(* IEC 61131-3 sources: ml2plc/examples/models/structured_text (part 2) *)

(* ---- test10_5k.st ---- *)
FUNCTION_BLOCK NeuralNetworkFB

VAR_INPUT
    input_data : ARRAY[0..4] OF REAL;
END_VAR

VAR_OUTPUT
    output_data : ARRAY[0..2] OF REAL;
END_VAR

VAR CONSTANT
    weights_0 : ARRAY[0..109] OF REAL := [-0.235502, 0.374035, 0.029982, 0.212839, 0.258987, -0.111841, 0.244708, -0.308510, 0.228488, 0.160992, 0.383056, 0.408669, -0.403928, -0.237195, 0.098766, -0.443759, -0.297004, -0.183076, 0.183679, -0.150052, -0.244251, -0.296679, 0.282903, -0.114856, -0.204128, 0.239042, -0.264883, 0.227759, -0.321238, 0.035633, 0.262893, -0.322360, -0.104940, 0.452904, 0.456325, 0.030485, -0.030166, -0.158633, 0.107382, -0.069652, -0.001856, -0.272029, -0.007177, -0.122300, 0.214300, 0.062439, 0.300184, -0.465629, -0.025417, -0.246331, 0.205803, 0.023458, -0.192963, -0.407002, -0.281354, -0.300315, -0.372232, -0.163916, -0.173461, 0.322071, 0.477836, 0.353802, 0.206684, 0.197231, 0.380607, 0.522870, -0.316586, 0.070922, 0.220201, 0.307742, -0.224637, -0.294651, -0.101183, 0.079923, 0.277857, 0.419958, -0.196677, -0.210945, -0.373816, 0.376826, -0.382129, -0.066666, 0.071888, 0.258300, -0.222091, 0.385427, -0.307561, -0.131309, 0.078177, -0.005495, 0.222825, -0.380124, -0.054474, -0.272398, -0.041792, 0.481035, 0.159107, 0.424615, 0.015366, 0.498193, -0.156387, 0.359789, 0.473488, -0.037305, -0.414866, 0.249786, -0.175640, 0.421966, 0.072167, -0.130746];
    bias_0 : ARRAY[0..21] OF REAL := [0.056635, -0.124397, -0.266900, -0.117066, -0.247369, -0.074615, -0.135742, 0.004444, -0.217433, -0.099763, 0.119883, -0.049615, -0.077851, -0.192466, -0.024998, 0.047683, 0.188981, -0.322050, 0.077329, -0.218410, -0.089648, -0.137956];

    weights_1 : ARRAY[0..483] OF REAL := [0.079049, -0.347925, 0.337554, -0.033540, 0.138506, 0.092452, -0.378136, 0.249819, -0.085962, 0.006912, 0.181653, 0.205352, -0.241950, 0.184875, 0.065784, -0.124519, 0.197723, 0.064407, 0.105942, 0.236089, 0.209018, 0.178479, 0.218949, -0.102088, -0.093211, -0.269140, -0.040398, 0.044989, 0.262907, 0.256715, -0.098784, 0.291057, 0.262021, 0.194998, -0.235076, -0.154412, -0.103262, 0.045983, -0.148590, -0.016494, -0.348144, 0.355634, -0.331634, -0.158894, 0.055906, 0.248997, 0.337778, -0.223945, -0.040168, 0.011934, -0.216079, -0.302210, -0.101061, 0.099673, 0.114095, 0.322268, -0.059129, -0.282656, -0.375054, 0.167089, -0.216769, 0.033994, -0.177784, 0.290487, -0.068697, 0.124034, 0.228402, -0.131462, -0.027060, 0.223431, -0.392828, 0.256138, -0.026546, 0.114889, -0.114368, 0.116107, -0.211801, 0.206436, 0.112972, 0.212281, -0.293026, -0.028103, 0.086852, -0.201455, -0.398612, 0.019805, 0.232748, 0.214277, -0.045702, -0.094083, -0.236141, 0.221850, 0.089407, -0.034819, -0.354278, 0.161435, 0.190216, 0.158098, 0.228709, -0.163889, 0.277531, -0.243516, 0.211692, -0.334966, 0.207670, 0.204391, 0.121696, -0.322424, 0.116413, -0.058254, -0.120124, -0.065694, 0.240498, -0.015988, -0.299633, 0.134494, -0.267642, -0.028926, 0.145824, -0.105526, -0.245366, -0.248820, 0.101097, -0.096212, -0.271919, -0.017597, -0.037329, 0.021210, -0.182566, 0.064379, -0.230258, -0.351002, -0.238026, 0.179422, 0.348074, -0.171654, 0.183988, -0.129054, -0.097976, 0.232130, 0.159159, -0.230301, 0.177287, -0.012360, -0.310712, -0.222650, 0.224205, -0.184178, 0.288744, 0.156265, -0.125907, 0.356347, -0.052188, -0.151564, -0.050163, -0.188746, 0.207031, 0.244088, 0.237136, -0.288542, 0.231177, 0.109337, -0.254618, 0.376183, -0.294310, 0.144768, -0.143697, -0.101113, -0.206989, 0.203110, 0.169697, -0.095264, 0.436408, 0.036662, 0.058565, -0.072889, 0.137062, 0.257720, -0.292869, 0.024309, -0.346628, 0.294436, 0.111847, 0.105722, 0.110252, 0.043315, 0.163461, -0.022499, 0.159847, 0.237663, 0.054308, 0.147833, -0.067078, -0.073643, -0.195978, -0.328734, -0.264882, -0.140460, -0.320087, 0.028090, -0.188938, -0.239834, -0.036262, 0.028815, 0.019727, -0.339510, -0.203977, -0.065838, 0.302599, 0.176075, 0.212229, -0.302148, 0.225811, 0.297823, -0.244519, 0.177079, 0.026356, 0.216062, 0.186228, -0.249791, -0.234059, -0.264074, 0.014307, -0.334354, -0.306848, -0.327795, -0.038307, -0.373215, -0.371131, -0.433094, -0.388753, -0.166083, -0.283418, -0.421748, -0.019741, -0.387288, 0.161504, 0.004465, 0.174149, -0.238579, -0.185134, 0.218629, -0.320004, 0.290548, 0.235413, -0.214184, -0.233729, -0.148321, -0.238665, -0.422416, -0.040923, 0.123327, -0.157409, -0.017170, 0.296382, 0.024681, -0.378978, 0.070786, -0.283947, -0.322869, 0.151345, -0.373138, 0.336530, 0.056313, -0.373142, -0.187809, -0.092519, 0.086954, -0.119277, -0.137913, -0.083906, 0.078384, -0.119447, -0.275883, 0.144350, 0.158292, -0.327999, -0.276656, 0.078429, -0.347799, 0.023557, -0.236602, -0.128356, -0.233653, 0.236965, 0.064413, 0.334948, 0.220999, -0.212444, 0.256759, -0.155419, 0.196652, 0.245904, 0.341258, 0.370730, 0.132005, 0.192064, 0.279513, -0.112169, 0.022927, -0.015424, 0.219870, 0.228535, 0.070248, -0.105873, -0.336300, 0.031945, 0.292533, 0.152411, -0.309550, 0.339161, 0.017188, 0.078137, -0.074693, -0.159284, 0.100658, 0.237390, -0.029114, 0.024597, 0.130221, -0.231880, 0.122851, -0.098909, 0.267768, -0.233404, -0.160178, 0.185329, 0.261339, 0.140867, 0.353704, 0.056444, 0.012285, -0.106170, 0.126114, 0.129954, 0.061448, -0.336865, -0.267193, -0.310728, -0.062605, -0.343586, -0.149127, 0.171627, 0.311902, -0.232079, -0.340220, -0.166417, -0.269893, -0.331138, -0.181041, -0.010986, 0.102309, -0.220985, -0.073660, -0.041843, -0.278722, -0.287776, 0.156741, 0.001601, -0.055916, 0.144559, -0.098055, -0.268363, -0.229689, -0.146128, -0.391409, 0.362549, -0.104388, 0.269200, -0.132739, -0.278950, -0.065837, -0.298305, 0.237254, 0.329178, 0.309923, -0.221904, -0.107192, -0.299514, 0.042806, 0.276688, -0.033415, 0.214313, 0.260739, -0.159463, 0.174015, -0.344592, -0.080061, -0.129057, -0.056141, -0.064048, 0.258323, 0.000715, -0.093780, -0.323654, -0.309229, -0.420076, -0.072576, -0.079502, 0.125576, -0.276341, -0.230562, -0.146622, -0.109113, 0.033652, -0.318611, -0.316500, -0.290675, -0.363042, -0.224463, -0.261462, -0.292973, 0.321195, -0.002662, 0.045876, -0.085935, -0.255877, 0.129174, 0.178717, 0.347154, 0.307062, -0.218534, -0.084984, -0.345322, 0.030590, -0.089027, 0.217998, -0.144714, -0.046250, -0.281607, -0.235275, 0.266412, 0.278757, 0.038723, 0.169535, 0.118446, 0.398865, 0.104389, -0.289460, -0.226774, -0.160745, -0.125390, 0.291478, -0.404079, 0.182954, -0.242632, -0.011222, 0.019191, -0.276508, 0.232760, 0.171934, -0.169843, -0.043784, -0.157749, -0.116427, 0.271703, -0.243017, 0.220278, 0.041874, 0.312852, -0.344001, 0.205275, 0.239192, -0.247240, 0.234474, -0.094469, -0.202707, 0.335269, 0.229963, 0.199586, -0.262707, 0.257955, -0.312206, -0.360458, -0.320586, 0.211516, 0.337735, 0.278487, 0.267389, 0.241000, -0.250274, 0.072497, 0.185405, 0.199016];
    bias_1 : ARRAY[0..21] OF REAL := [-0.155419, -0.267332, -0.021124, -0.086635, -0.086491, 0.106494, -0.081331, -0.149528, 0.128646, 0.006162, -0.052589, -0.175140, 0.004669, -0.158592, -0.001915, -0.165681, -0.032700, -0.202270, -0.109741, 0.031299, -0.051547, 0.080420];

    weights_2 : ARRAY[0..483] OF REAL := [-0.082935, 0.327544, 0.254661, -0.021772, 0.201947, 0.305412, 0.081183, 0.318496, 0.143632, -0.205671, 0.060881, -0.296683, 0.233208, -0.132674, -0.267633, 0.297422, -0.148609, 0.024956, -0.328323, 0.249083, 0.322392, 0.251571, -0.079101, 0.041405, -0.094899, -0.052703, -0.228929, -0.173477, 0.309499, -0.298324, -0.328228, 0.191809, 0.211639, 0.175227, -0.291024, -0.241829, -0.227845, 0.359827, -0.173025, -0.185764, -0.281586, -0.131694, -0.345628, -0.036727, -0.163816, -0.334208, -0.132535, 0.173024, 0.224584, -0.343964, -0.252016, -0.342804, 0.081973, 0.110123, 0.056545, -0.049518, 0.216609, -0.092255, -0.220284, 0.153317, -0.178284, 0.077126, -0.381740, 0.041970, 0.118417, -0.290151, 0.228592, -0.343728, 0.081173, 0.186181, 0.042570, -0.032074, -0.347268, 0.039175, 0.205202, -0.321549, -0.104232, -0.302562, -0.251374, 0.314923, 0.045477, -0.033431, -0.386075, 0.012686, 0.125798, -0.210791, -0.393972, -0.352663, 0.300682, 0.233090, 0.060526, 0.143590, 0.215293, 0.298667, 0.050667, 0.195947, 0.172492, 0.286427, -0.276380, -0.344604, -0.295523, -0.000179, 0.252037, 0.155288, 0.180119, -0.282181, -0.368783, 0.259566, -0.153441, -0.230622, 0.294233, -0.076799, -0.375942, -0.345544, -0.163923, 0.044519, -0.319325, 0.221346, -0.132698, -0.127449, 0.026434, -0.149147, -0.076145, -0.306095, -0.253755, -0.312573, 0.021093, -0.181651, -0.290607, 0.083633, -0.150752, 0.006249, -0.298933, 0.333710, 0.325536, -0.222120, 0.278292, 0.100666, -0.085205, -0.356550, 0.185289, 0.084207, 0.177925, -0.233948, -0.031037, 0.031882, -0.276591, -0.200347, -0.265831, -0.171206, -0.121855, -0.272616, 0.106950, 0.267811, 0.144345, -0.141822, 0.314253, -0.139761, 0.326825, -0.240426, 0.203541, 0.224520, -0.346032, 0.054895, 0.171094, 0.049029, -0.116277, -0.143705, 0.283372, -0.025292, -0.333692, -0.302754, 0.050393, 0.194249, -0.151961, 0.190338, -0.155851, -0.230143, -0.286497, 0.344899, 0.024594, 0.079224, -0.023155, 0.030636, 0.121751, 0.115104, -0.101916, -0.335504, -0.111129, -0.103364, 0.171968, -0.336117, 0.022877, 0.127892, -0.135068, -0.122467, -0.396051, 0.145917, -0.006995, 0.381155, -0.271586, 0.211470, 0.293431, 0.054489, 0.267433, 0.043922, -0.036805, -0.139896, -0.059831, 0.220703, 0.157794, -0.123315, -0.004200, -0.389434, -0.119506, 0.234269, -0.144908, -0.325883, 0.023704, -0.203639, 0.025667, 0.011748, 0.296067, 0.257535, 0.341761, 0.013412, -0.246624, -0.031834, 0.012090, -0.022462, 0.387307, -0.315927, 0.135532, -0.106146, -0.208187, -0.077365, 0.210223, -0.164290, 0.117905, -0.141453, -0.062069, 0.078166, 0.197727, -0.315830, -0.359223, -0.000416, 0.153591, 0.293815, -0.088260, -0.024230, 0.338556, 0.085211, -0.209096, 0.270740, 0.266294, 0.103243, 0.280570, 0.004210, 0.174240, 0.393157, -0.136366, -0.322978, -0.000434, 0.228373, -0.258511, 0.179665, -0.222202, 0.114817, 0.119143, 0.073947, -0.261211, 0.292751, 0.027004, -0.307591, 0.184837, -0.129084, -0.067745, -0.033641, 0.037630, -0.078543, -0.085143, -0.098848, -0.030430, 0.187926, -0.058864, -0.145514, -0.132123, 0.143235, 0.158167, 0.062374, 0.066104, 0.019079, 0.251746, -0.122901, 0.164780, -0.194877, 0.219013, -0.242652, -0.214676, -0.076353, -0.249113, 0.221838, 0.199792, 0.181832, -0.230836, -0.109779, 0.133959, -0.036438, -0.249530, 0.199512, -0.095072, 0.093821, 0.071035, 0.061617, -0.279793, -0.201789, 0.187455, 0.018947, 0.050322, 0.008108, -0.046991, 0.306518, -0.327390, -0.138280, 0.116354, -0.106726, 0.207402, -0.069084, -0.132325, -0.310824, -0.166095, 0.230069, -0.389367, 0.254957, 0.026655, -0.361433, -0.138050, 0.059506, 0.152043, -0.028680, 0.287269, 0.153620, -0.085093, 0.109935, -0.100580, -0.031819, 0.185861, 0.392915, -0.032841, 0.080074, 0.306054, 0.027516, -0.379458, 0.256309, -0.393753, 0.001235, -0.319371, 0.251579, 0.125351, 0.073606, -0.082433, -0.161256, -0.069119, -0.211557, -0.294755, -0.267203, -0.224041, -0.309678, -0.351013, 0.121915, -0.248513, 0.271583, 0.124953, 0.201983, 0.198783, 0.099953, 0.131763, -0.286613, -0.229959, -0.150241, 0.379902, -0.322958, 0.278217, 0.239573, -0.287928, 0.336981, 0.176765, 0.110885, 0.159063, 0.293586, 0.322831, -0.086323, -0.214025, -0.030494, -0.146554, 0.020220, 0.070352, -0.005592, 0.164585, -0.044105, -0.015679, 0.194617, 0.231574, -0.021186, -0.312370, 0.146685, 0.363802, -0.404818, 0.063827, -0.091208, 0.104540, 0.112544, 0.225414, 0.426742, 0.164169, -0.015709, 0.332852, 0.015972, 0.245230, -0.030557, -0.123999, -0.129163, -0.298851, -0.172933, 0.228824, 0.231744, 0.039497, 0.270405, -0.303923, 0.058437, -0.216858, 0.034896, 0.123225, -0.159160, -0.288073, -0.040648, -0.108659, -0.092023, 0.054152, -0.387218, 0.163232, 0.184591, 0.243524, -0.138134, -0.341152, 0.046506, -0.346441, -0.281175, -0.387726, 0.123238, -0.300494, 0.237686, -0.045294, -0.331050, -0.130853, -0.231359, 0.222539, -0.205569, -0.347141, -0.176774, 0.238876, -0.010123, -0.432586, -0.172873, -0.266623, -0.267432, -0.083994, -0.348342, 0.095161, -0.382534, -0.225168, -0.199141, 0.018341, -0.198148, 0.198510, 0.236356, -0.289449, 0.075354, -0.175895, -0.114134, 0.042550, -0.277356, -0.088906, -0.080386];
    bias_2 : ARRAY[0..21] OF REAL := [-0.132522, -0.027953, -0.156794, -0.173189, -0.073986, -0.111488, -0.182651, -0.158691, -0.185292, -0.282737, -0.305989, -0.185168, -0.048515, -0.036091, -0.075189, -0.198026, -0.136586, -0.106037, -0.051125, -0.059318, -0.072963, -0.191347];

    weights_3 : ARRAY[0..483] OF REAL := [-0.070963, 0.130692, -0.269850, 0.140810, -0.058719, 0.300814, 0.273362, -0.241552, 0.052187, 0.139223, -0.312618, 0.302189, 0.204637, 0.280806, 0.249241, 0.239799, -0.030181, 0.299634, -0.158570, -0.240536, 0.039247, -0.093849, -0.069672, -0.110026, 0.104300, 0.006270, -0.065404, -0.061827, 0.137584, 0.113450, 0.233291, 0.031230, -0.224060, -0.007959, -0.009959, -0.207101, 0.114770, 0.173167, 0.251814, -0.079727, -0.083826, -0.260188, -0.310279, 0.104744, 0.107125, 0.207032, -0.318996, 0.159255, 0.034373, 0.237722, 0.033715, -0.121734, -0.224087, 0.206738, 0.059584, 0.299180, 0.068442, -0.156955, 0.145228, -0.100454, -0.225023, -0.273292, 0.280308, 0.093051, -0.354356, 0.032969, -0.196454, -0.130776, -0.143975, 0.084145, 0.129234, -0.034169, 0.310125, -0.085513, 0.109817, -0.218289, 0.008993, 0.240534, 0.285099, -0.293260, -0.239596, -0.215456, 0.128503, -0.107708, 0.160487, 0.124243, 0.151635, 0.304328, -0.107218, 0.270742, 0.065129, 0.166662, -0.046038, -0.054938, 0.022022, -0.104007, 0.128583, -0.099885, -0.048699, -0.033328, 0.088990, -0.288285, -0.222791, -0.051723, 0.290322, -0.252797, -0.030634, -0.152525, -0.258451, -0.281153, -0.326554, 0.119863, 0.153369, -0.265971, -0.090043, -0.078578, -0.240882, 0.180207, -0.119918, -0.152555, 0.055530, -0.298942, 0.266564, 0.208837, 0.267554, -0.040036, 0.109819, -0.096050, 0.008369, 0.201054, -0.250575, -0.002223, 0.202218, -0.367155, 0.007635, -0.135730, 0.257787, 0.180198, -0.007797, 0.275950, -0.072008, -0.293672, -0.178437, 0.401395, -0.186727, -0.097857, -0.149188, 0.348780, -0.104043, -0.373279, -0.236812, 0.269518, -0.374350, -0.170940, 0.198624, -0.188143, -0.180487, 0.265100, 0.173555, -0.264366, 0.314584, -0.034188, 0.151072, 0.251236, 0.078866, 0.159427, -0.330060, 0.000300, 0.302961, -0.200148, 0.277048, 0.005095, 0.025485, 0.099432, 0.204978, 0.188643, -0.361716, 0.325723, 0.024829, 0.213730, 0.003386, -0.335407, 0.036445, 0.098838, 0.141934, -0.230750, -0.146777, 0.121431, 0.263906, -0.350266, 0.249431, 0.082268, 0.020137, -0.307357, -0.075153, -0.238399, 0.301961, -0.247934, -0.354909, 0.170639, -0.290637, 0.243225, 0.205882, -0.291780, 0.061915, 0.122856, 0.109378, 0.041539, 0.229212, 0.063917, -0.310349, 0.081571, -0.230271, -0.135369, 0.252606, 0.291976, 0.217874, 0.171455, -0.123281, 0.338451, 0.237522, -0.016180, 0.009211, -0.150392, 0.120245, -0.128392, 0.362670, 0.229386, 0.139791, 0.086210, -0.120099, -0.257756, 0.336282, -0.184179, 0.061028, 0.268711, 0.297470, 0.006473, -0.155874, 0.119006, -0.147172, 0.338455, -0.306829, 0.201802, -0.245255, -0.003989, -0.056203, -0.371497, 0.294629, -0.354312, 0.274458, -0.369053, 0.303723, -0.231104, 0.162307, -0.146596, -0.247671, 0.209516, 0.096599, -0.220339, 0.081374, 0.282433, 0.217082, -0.143945, 0.186003, 0.041982, -0.257384, 0.261132, 0.099202, 0.017216, -0.307124, 0.006945, -0.221664, -0.224805, -0.289980, 0.210305, -0.045192, -0.260953, 0.350597, -0.285064, -0.195511, -0.178267, 0.137539, -0.023689, -0.244267, -0.325062, 0.158579, -0.252519, -0.111991, -0.104875, -0.051395, -0.387023, 0.105685, 0.065664, -0.182484, 0.126195, 0.006960, -0.108073, 0.108834, 0.004119, -0.109705, 0.263873, -0.022458, -0.322233, 0.255739, 0.247398, -0.303781, 0.236973, -0.227161, 0.326930, -0.032857, 0.324233, -0.316049, -0.196805, 0.324190, -0.102829, 0.202962, -0.249527, 0.174379, 0.017646, 0.136594, 0.068535, -0.073554, -0.053696, 0.094891, -0.002721, -0.029553, 0.298469, 0.228519, 0.132958, -0.280243, 0.348791, -0.244033, 0.180527, 0.291389, -0.227724, -0.080778, 0.026035, -0.349332, 0.025376, 0.323342, -0.168050, 0.170721, 0.141696, 0.287412, 0.303008, -0.297372, -0.231378, -0.327177, 0.245814, -0.157496, 0.305786, 0.023815, 0.194373, 0.042962, 0.247734, -0.017229, -0.287956, -0.153367, -0.265115, -0.157484, -0.254438, -0.322820, 0.274838, 0.147736, 0.285888, 0.231649, 0.174032, 0.175934, 0.271467, 0.084399, -0.019627, 0.341451, 0.178289, 0.095685, 0.351044, -0.236451, 0.029438, 0.124888, 0.252756, -0.024477, -0.167562, 0.122333, -0.363672, -0.280869, 0.350745, 0.008932, -0.056523, 0.321664, 0.072688, -0.308330, -0.056758, -0.378707, 0.016178, 0.157754, 0.280456, -0.072451, 0.008635, 0.056400, -0.027879, -0.023298, 0.293456, 0.073344, 0.066010, 0.107840, 0.056185, 0.092087, -0.038662, -0.081590, 0.048914, -0.042117, -0.050272, 0.235561, 0.097758, 0.159443, -0.282414, -0.070700, 0.045638, -0.235297, 0.028984, 0.315669, -0.365402, -0.397538, 0.246604, -0.370567, -0.264243, -0.335273, -0.267622, -0.027876, -0.045249, 0.256983, -0.282323, -0.190901, 0.327641, 0.120722, 0.244446, -0.099077, -0.093646, 0.064414, 0.091739, 0.072448, -0.174493, -0.268327, -0.043659, 0.362111, -0.362721, -0.062207, 0.237062, -0.289300, 0.262508, 0.024987, 0.186755, -0.206446, 0.190574, -0.002648, 0.135858, 0.070928, -0.079544, 0.202876, -0.090191, 0.004004, -0.238061, 0.012142, 0.281664, -0.076509, 0.294768, -0.090052, 0.135075, -0.127598, 0.167098, -0.091762, -0.329548, 0.091189, 0.115618, -0.156032, -0.058680, 0.028823, -0.335428, -0.196004, -0.384244, 0.121939, 0.289472, 0.326180, 0.182819];
    bias_3 : ARRAY[0..21] OF REAL := [-0.071660, -0.155321, 0.017151, -0.127591, -0.172606, -0.117057, -0.059306, -0.195838, -0.144730, -0.026066, -0.113688, -0.103356, -0.071603, -0.088934, -0.090114, -0.112454, -0.226730, -0.045391, -0.072792, -0.260438, -0.183089, 0.010589];

    weights_4 : ARRAY[0..483] OF REAL := [0.285340, 0.124708, 0.032434, -0.070546, 0.323896, 0.314783, 0.156508, 0.049337, -0.257855, 0.060797, 0.225259, -0.343727, -0.305054, 0.264680, -0.259098, 0.100738, 0.130620, 0.155558, 0.180438, 0.018363, 0.292032, -0.186949, 0.344697, 0.008839, 0.278729, 0.329124, -0.104647, -0.116247, 0.185435, 0.117228, 0.259561, 0.191473, 0.044427, 0.156030, 0.179480, -0.030503, -0.192425, 0.146114, -0.011534, -0.101514, -0.309830, 0.128590, -0.175476, 0.248233, 0.118166, 0.298943, 0.153585, -0.190505, 0.132242, 0.343228, -0.279652, 0.281808, -0.327119, 0.270119, -0.109654, 0.002895, -0.279353, 0.043761, -0.332060, 0.395426, -0.111156, 0.107962, 0.175226, -0.119038, -0.013641, -0.319853, 0.046963, 0.112984, -0.269099, -0.181680, 0.214857, -0.147116, -0.297881, -0.019060, 0.276537, -0.278688, 0.238607, -0.308053, 0.261947, -0.138666, 0.200434, -0.093892, 0.284911, -0.105623, -0.239891, 0.138511, 0.290045, -0.068706, -0.251814, -0.103389, 0.111106, 0.140267, -0.164758, -0.073620, 0.259873, -0.134675, 0.299443, 0.210446, -0.242414, -0.228769, 0.044735, -0.190339, 0.173803, 0.201277, 0.265555, 0.281608, 0.303993, 0.193458, -0.376399, 0.041768, 0.186414, -0.208191, 0.224658, 0.244820, -0.301394, -0.104093, -0.056840, -0.260437, -0.086111, -0.262008, -0.223552, -0.035133, -0.265831, 0.200115, 0.190150, -0.178191, -0.040832, -0.155468, 0.030926, 0.214046, -0.403207, 0.052822, 0.028208, 0.120102, 0.253822, 0.331983, 0.290159, 0.098311, -0.140303, -0.032536, -0.111903, -0.128369, -0.221021, 0.089680, -0.325587, 0.173947, 0.305488, 0.073691, -0.126267, -0.277542, 0.047927, -0.300922, 0.067113, 0.248527, 0.312853, 0.291413, -0.139322, 0.196262, 0.167906, 0.067655, -0.124497, 0.228796, 0.270043, 0.073319, -0.028912, -0.351353, -0.142426, -0.113276, 0.167101, -0.152871, 0.244701, -0.179737, 0.029928, 0.012332, 0.117012, 0.232886, 0.253417, 0.277782, 0.356720, -0.053588, -0.219849, 0.161095, 0.282162, -0.044447, 0.252406, -0.317867, -0.064759, 0.199853, 0.266236, -0.227075, -0.160522, -0.131642, -0.162327, 0.242400, -0.291850, 0.233357, 0.312205, 0.189678, -0.020536, -0.225512, -0.125560, 0.207247, 0.018774, -0.058509, 0.248546, 0.122879, -0.273556, 0.018504, 0.172931, 0.099942, -0.264318, 0.265185, 0.060279, -0.088737, -0.239243, 0.070758, -0.205583, -0.223837, -0.322970, -0.039312, 0.150358, 0.155740, 0.063867, -0.103831, 0.206850, -0.140231, 0.093940, -0.130947, -0.212310, 0.039814, 0.196195, 0.119526, -0.220981, 0.317267, 0.176579, -0.245296, 0.310520, 0.186219, 0.021436, 0.252485, 0.043407, -0.184534, -0.166159, -0.289449, -0.134246, 0.185497, -0.332515, -0.300164, 0.071231, -0.007877, -0.341469, -0.313808, 0.299587, -0.332565, -0.029276, 0.234033, 0.075816, 0.123334, 0.056343, 0.319063, -0.170227, 0.335196, -0.096163, 0.127576, -0.157330, -0.175745, 0.015556, -0.197033, -0.041917, 0.079742, -0.068899, -0.310613, -0.286623, -0.110462, 0.200041, -0.298751, 0.364553, 0.288485, -0.233971, -0.259451, 0.181023, -0.149220, 0.321499, 0.380083, 0.276357, -0.289341, -0.177815, 0.288891, -0.267010, -0.292728, -0.133176, -0.181918, 0.164240, -0.336144, -0.136582, 0.188441, -0.230141, 0.059835, 0.162013, 0.139585, 0.128726, 0.179736, -0.163349, -0.173248, 0.117859, 0.267253, 0.188233, -0.167903, -0.029504, -0.175437, -0.056729, 0.326573, 0.229124, 0.135776, 0.111830, 0.020920, -0.171492, 0.184173, 0.152547, -0.124838, 0.301794, -0.229966, -0.198163, -0.079993, 0.141797, 0.374755, 0.295944, 0.013124, 0.331928, -0.187327, 0.253732, -0.390516, -0.187737, -0.190255, -0.135552, 0.269689, -0.231294, -0.273829, -0.410815, 0.303615, -0.390827, -0.089264, 0.069898, -0.010489, 0.192258, 0.338348, 0.312908, -0.061972, -0.199711, -0.265956, -0.156552, 0.030330, 0.124526, 0.085226, -0.238105, 0.173442, -0.125368, 0.049648, -0.135100, -0.202399, 0.122846, 0.029544, 0.246183, 0.058490, 0.079692, 0.026235, 0.249573, -0.011999, -0.317708, 0.127146, 0.336527, 0.310867, -0.048611, 0.119099, -0.114378, 0.035412, 0.330085, -0.036438, 0.320118, -0.343053, 0.206974, -0.022545, -0.167291, 0.319224, 0.290293, 0.224596, -0.014116, -0.058974, -0.236342, -0.037211, 0.134922, 0.205024, 0.092058, -0.171377, 0.104657, 0.254821, -0.256170, -0.017548, 0.152745, 0.104539, 0.059229, 0.033481, -0.330303, 0.021580, -0.159210, -0.243931, 0.147111, 0.204359, -0.311978, 0.063528, -0.222022, 0.075310, 0.007856, -0.322708, 0.235170, 0.193480, 0.150068, 0.049194, 0.296921, 0.169293, 0.080050, 0.114132, -0.318059, 0.136174, 0.304245, -0.033880, 0.149083, -0.387539, -0.199142, 0.110489, 0.316280, -0.034479, -0.189814, 0.382408, -0.125453, 0.230444, -0.158843, 0.236897, 0.009293, 0.044525, -0.105016, 0.261944, -0.117140, -0.165268, 0.197458, 0.272622, 0.155061, 0.071731, 0.222820, -0.357453, -0.300762, 0.178104, 0.063046, 0.029061, 0.109896, -0.131855, 0.189788, 0.317413, 0.165292, 0.141550, -0.035790, 0.214812, -0.151208, -0.253156, -0.011525, 0.049784, -0.232897, -0.208622, 0.320459, -0.262409, -0.150645, -0.354825, -0.359394, 0.312819, -0.222176, -0.005476, 0.136215, 0.165142, -0.004936, -0.272071, -0.027402, -0.132006, 0.106643, 0.047964];
    bias_4 : ARRAY[0..21] OF REAL := [-0.135631, -0.059973, -0.057355, -0.076233, 0.006988, -0.120337, -0.087401, 0.015224, -0.113106, -0.057927, 0.018011, -0.072078, -0.149866, -0.087133, -0.147846, -0.034441, -0.159101, 0.011132, -0.071134, -0.224402, -0.068134, -0.157693];

    weights_5 : ARRAY[0..483] OF REAL := [0.295786, -0.183677, -0.194963, -0.012476, 0.325160, -0.248307, -0.032719, 0.350695, -0.041984, -0.039824, -0.123213, 0.205041, 0.309413, 0.054617, 0.214864, -0.199095, 0.080945, 0.081340, 0.340758, 0.125757, -0.127943, 0.020536, -0.120914, -0.324866, -0.278909, -0.132589, 0.182998, 0.127864, -0.188677, 0.320486, 0.075749, 0.128434, -0.269198, 0.251693, 0.202992, -0.070689, -0.321505, -0.110830, 0.177488, 0.005186, -0.090039, -0.103660, 0.047995, 0.322856, 0.050662, -0.275122, -0.256324, 0.226610, -0.236704, 0.086131, -0.252113, 0.113707, -0.235460, -0.221253, 0.149488, -0.025197, 0.269246, -0.017756, 0.058502, 0.371721, -0.196094, 0.362806, 0.214972, -0.061153, -0.032495, -0.314799, -0.312536, 0.112301, 0.070488, -0.192138, 0.325300, -0.176772, -0.138474, 0.167194, 0.276014, 0.164868, -0.329372, 0.161283, 0.263398, 0.348368, 0.131874, 0.256534, 0.220644, 0.356568, -0.372424, -0.079733, 0.245019, -0.083489, 0.032426, 0.273998, -0.099620, 0.334057, -0.333146, 0.270987, -0.309939, 0.263709, 0.294746, -0.057703, 0.302831, -0.138752, -0.018732, -0.082801, 0.181588, 0.387898, -0.143796, -0.245350, -0.111428, 0.273398, -0.205308, 0.206082, -0.083602, 0.318211, 0.065567, 0.083594, 0.122775, -0.147773, -0.024361, -0.259743, -0.125003, -0.113708, 0.096325, -0.227137, -0.239484, -0.305946, -0.199726, 0.214570, 0.279476, 0.173012, -0.116649, 0.049696, 0.257520, -0.285520, -0.010751, 0.069927, -0.272949, -0.103210, 0.165375, -0.313160, -0.173223, -0.020450, -0.251738, -0.281475, 0.090597, -0.181312, -0.068716, 0.319115, -0.141168, 0.254548, -0.328429, -0.245433, 0.352490, 0.231462, 0.285700, 0.282915, -0.137530, -0.104165, -0.082240, 0.206955, 0.083898, 0.217600, 0.253571, 0.174800, 0.183454, 0.322473, 0.261781, -0.203370, -0.296975, -0.157250, -0.340946, 0.003344, -0.080648, -0.376684, -0.321230, 0.166949, -0.073823, -0.017077, 0.176695, 0.140181, -0.294874, 0.050852, 0.294428, -0.371712, -0.252088, -0.172532, -0.275701, 0.092976, -0.231732, -0.004416, -0.116009, 0.069547, 0.212635, -0.181009, 0.070041, -0.202499, -0.018228, -0.060812, -0.078127, 0.228379, -0.004143, -0.275358, -0.216025, -0.286885, -0.352893, -0.352714, 0.259360, 0.202026, 0.162057, -0.176679, 0.092397, 0.023471, -0.285262, 0.093350, -0.120427, -0.051339, 0.055293, 0.102931, 0.051467, 0.047042, 0.154991, 0.210889, -0.078130, -0.199765, 0.058239, -0.237824, -0.298788, -0.032308, -0.129379, 0.059440, -0.266609, -0.265022, 0.095976, -0.008170, -0.116087, 0.065678, -0.372756, -0.027756, 0.095709, 0.096379, 0.108798, 0.337119, 0.115758, 0.167660, -0.138890, -0.257222, -0.291318, 0.247571, -0.072634, 0.147559, 0.266334, 0.316704, -0.039131, -0.106945, 0.096779, -0.239564, 0.178228, 0.025796, 0.318465, 0.053781, 0.038663, 0.212693, -0.264130, 0.269332, 0.144596, -0.020079, -0.142040, 0.345830, 0.294463, -0.284632, 0.303159, -0.055051, -0.175444, -0.004635, 0.245131, 0.347638, -0.363994, 0.354520, 0.345105, -0.124907, 0.175329, -0.252487, 0.218221, -0.288665, -0.185736, 0.228403, -0.007983, -0.328992, 0.186340, -0.052072, 0.177608, 0.313255, 0.341282, 0.124264, 0.290080, -0.306797, 0.156603, -0.040627, 0.199176, 0.010949, 0.298901, -0.003477, -0.319152, -0.160251, 0.347125, 0.120863, -0.057133, -0.108501, -0.101377, -0.416108, -0.256034, 0.345127, 0.075900, 0.077434, -0.327498, 0.300395, 0.263323, 0.033518, -0.098224, 0.313559, 0.057109, 0.268897, -0.168572, 0.104852, -0.090507, -0.022958, -0.129505, 0.155949, 0.177589, -0.299684, 0.260695, 0.235179, -0.239140, 0.294636, 0.220173, 0.246848, -0.143859, -0.015503, -0.201013, -0.266079, -0.365497, 0.150639, -0.316233, 0.212970, 0.118881, 0.095540, -0.351161, 0.340327, -0.127609, -0.241068, -0.102025, -0.150887, -0.175063, 0.246760, 0.105128, 0.231438, -0.316038, -0.021280, 0.116366, 0.239533, -0.099675, -0.273935, 0.215278, -0.305493, 0.128501, -0.320110, 0.106418, -0.158291, 0.330269, -0.199709, 0.150859, 0.201374, 0.302986, 0.293814, 0.145793, -0.063855, 0.274164, -0.267782, -0.059552, -0.110310, 0.072082, 0.004304, -0.273820, 0.136195, -0.059846, 0.195179, -0.050319, 0.304967, 0.198983, 0.034801, -0.056669, -0.155134, 0.130003, -0.334066, -0.237327, 0.123767, -0.148630, 0.246949, 0.120109, 0.292648, 0.000135, -0.103384, -0.177117, 0.295904, 0.207313, -0.287970, -0.242404, 0.338894, 0.042522, 0.219264, -0.256873, 0.330269, 0.076745, -0.114580, 0.348135, -0.350177, 0.027450, -0.325224, -0.325608, -0.211409, 0.059599, 0.340820, 0.188550, 0.233273, 0.094421, 0.349525, -0.377160, -0.123297, 0.174766, 0.226045, -0.241743, 0.226283, 0.133306, -0.155922, -0.025345, 0.239190, -0.272052, -0.104206, 0.289481, 0.028963, -0.240904, 0.241072, 0.242253, 0.138540, -0.026430, 0.274806, 0.104138, -0.137693, -0.227110, -0.266070, -0.220316, -0.028174, 0.039213, 0.123646, -0.309178, 0.351024, -0.062718, -0.049403, -0.330493, -0.289171, 0.330889, -0.117402, 0.042765, 0.267620, -0.067596, 0.288371, 0.220475, 0.220831, -0.340022, 0.319252, 0.148340, 0.175661, -0.326485, -0.196901, -0.323719, 0.177351, 0.327086, -0.223148, -0.289504, -0.142860, 0.270837, -0.283047, 0.248922, 0.065004, 0.196505, 0.016435];
    bias_5 : ARRAY[0..21] OF REAL := [-0.108748, -0.148790, -0.169750, -0.063060, -0.136281, -0.015090, -0.123394, -0.066572, -0.039855, -0.071659, -0.057859, -0.022162, -0.013096, 0.008857, -0.085195, -0.048427, -0.108942, -0.040683, -0.190474, -0.056512, -0.080564, -0.103133];

    weights_6 : ARRAY[0..483] OF REAL := [0.000226, -0.317295, 0.216378, 0.057080, -0.202799, -0.323463, 0.023792, 0.338432, 0.298338, 0.317400, -0.317865, 0.078150, 0.384632, -0.027240, -0.017339, 0.269326, 0.319771, 0.334347, 0.190047, 0.099784, 0.205733, -0.312326, -0.368901, -0.218586, -0.228075, -0.164128, 0.039126, 0.218889, 0.162654, -0.303201, 0.310733, -0.069633, -0.206399, -0.129089, 0.297279, -0.100493, 0.127634, 0.300330, -0.293205, -0.054581, 0.101621, 0.336318, -0.132218, -0.066936, 0.140740, 0.178458, 0.130402, 0.131257, 0.255337, 0.201279, 0.243607, -0.065641, -0.131974, 0.340401, -0.010297, 0.265703, -0.124207, 0.214099, 0.022107, 0.173648, -0.208697, -0.270572, 0.009770, 0.212335, -0.354614, -0.045055, 0.165315, 0.017672, -0.318987, 0.231848, 0.269806, 0.099017, -0.143021, 0.106106, -0.216196, 0.273588, -0.224648, 0.142580, 0.200526, 0.265644, 0.123300, -0.310863, -0.186073, -0.005301, -0.031029, 0.105821, 0.109991, 0.036367, 0.234359, -0.163618, 0.002875, 0.207435, -0.314401, -0.193510, -0.247448, -0.199878, 0.294441, -0.266737, -0.005412, 0.041695, 0.304971, -0.066309, 0.183374, 0.292544, 0.211918, 0.008088, -0.061046, 0.278876, -0.244374, 0.266993, -0.198886, -0.252755, -0.341022, 0.338738, 0.203630, -0.031769, -0.112598, -0.186243, 0.167516, -0.167116, -0.080773, -0.135911, -0.320650, -0.086755, 0.285659, -0.164102, -0.094649, -0.141913, -0.132173, 0.067571, -0.175439, 0.052214, -0.132600, -0.148676, 0.135414, 0.079742, 0.343727, -0.268583, 0.046536, -0.118576, -0.221659, -0.323323, -0.336178, 0.243220, 0.128952, 0.152764, 0.078811, 0.351498, -0.239569, 0.165505, -0.024044, 0.266859, 0.370605, 0.279072, -0.163479, -0.210041, 0.226665, -0.178820, -0.234092, -0.373663, 0.178702, -0.064686, -0.004987, 0.268417, -0.358069, 0.029933, 0.040636, 0.182228, -0.373903, 0.005117, -0.349272, -0.113149, 0.225492, -0.133442, -0.051294, -0.018002, 0.197050, 0.093261, -0.060199, -0.240084, -0.323600, -0.116586, -0.101561, -0.328429, 0.039808, 0.173261, 0.258801, -0.230536, 0.156868, 0.167958, 0.180630, 0.068932, 0.183490, -0.232715, 0.319523, -0.030165, 0.268916, -0.130119, -0.207572, -0.332430, 0.265373, 0.062630, 0.265256, -0.156984, 0.326607, 0.021322, -0.019128, 0.221891, -0.128364, 0.116103, 0.177029, -0.267860, 0.109979, -0.309246, 0.252922, -0.350642, -0.288182, -0.049970, -0.216187, -0.230961, 0.268968, 0.039614, 0.049786, -0.317580, -0.353649, 0.144283, 0.278989, 0.044691, -0.000908, 0.165982, 0.111109, 0.059366, -0.204298, 0.086981, 0.328572, 0.238897, 0.294931, -0.250349, 0.384107, 0.110253, -0.159390, 0.191167, -0.172712, 0.133281, 0.207976, 0.018425, -0.090964, -0.077157, -0.285751, -0.247010, -0.053044, 0.026488, 0.242353, 0.300082, -0.279388, -0.222664, -0.346127, 0.340803, -0.100380, -0.196143, 0.303490, -0.273116, 0.019828, -0.124140, -0.262377, -0.211975, -0.060136, 0.245106, -0.049269, 0.348477, -0.354285, -0.234125, 0.071312, 0.039700, -0.045883, -0.159054, -0.004032, 0.035592, -0.106654, -0.184796, 0.144523, -0.179010, -0.021851, -0.359204, 0.136350, 0.228865, -0.233354, -0.334930, 0.146104, -0.287607, 0.191988, -0.192312, 0.278091, 0.171834, 0.093334, 0.127515, -0.204526, -0.346142, -0.176639, -0.188276, -0.158835, -0.342356, -0.224487, -0.131235, 0.125573, -0.285720, 0.275527, -0.125556, 0.220248, 0.056655, -0.112171, 0.304454, 0.128032, -0.309690, 0.156499, 0.047870, -0.121099, -0.265502, -0.043752, -0.269809, 0.048821, -0.161326, -0.061197, 0.036180, 0.028718, 0.264457, -0.194159, 0.322621, 0.328862, -0.113418, 0.071989, 0.349598, 0.408608, 0.334123, -0.192248, -0.014832, -0.294235, 0.130985, 0.227693, 0.440277, -0.353239, -0.102317, -0.180273, -0.130511, 0.232047, 0.299197, -0.326744, -0.196980, 0.051820, 0.085804, -0.175758, -0.070172, -0.007210, -0.222703, 0.222136, -0.352179, 0.039003, -0.051871, 0.161134, 0.320371, 0.227055, 0.306207, 0.040361, -0.017315, -0.309185, -0.272377, 0.085801, 0.270702, -0.030839, -0.322727, 0.124320, 0.032711, -0.169684, 0.191543, 0.148049, -0.141451, 0.322499, -0.297789, 0.150025, -0.121595, 0.072254, 0.132663, -0.252835, 0.051657, 0.195058, -0.136630, 0.153772, 0.254306, -0.142885, -0.251978, 0.341934, 0.174483, 0.143433, -0.091235, 0.069374, -0.077009, -0.009924, -0.272147, -0.160586, 0.118563, 0.258597, -0.311079, 0.261532, -0.240238, 0.044522, 0.098922, -0.013241, -0.262968, -0.346938, -0.242160, -0.368006, 0.341509, 0.271318, 0.118895, -0.272983, -0.080571, 0.106451, 0.101326, 0.216311, -0.136889, -0.039425, -0.162027, -0.078030, 0.280973, -0.033615, -0.284168, -0.057450, 0.318053, -0.012656, -0.286653, 0.359645, -0.116870, -0.062116, -0.283753, 0.112345, -0.293851, 0.323846, 0.088058, 0.189790, -0.084003, 0.174591, 0.129663, 0.126038, -0.371679, 0.073706, 0.142749, 0.302681, -0.145627, 0.025066, 0.225651, -0.084100, -0.290841, -0.073780, -0.190614, -0.185107, -0.142582, 0.182609, 0.325726, -0.120137, -0.285171, 0.291144, 0.146397, 0.060717, 0.025991, -0.300234, -0.300862, -0.089209, -0.021209, 0.321965, -0.024053, 0.356330, 0.091753, -0.129269, 0.013336, -0.155416, 0.021223, 0.107530, -0.338468, -0.062504, 0.311934, 0.179257, -0.086443, -0.180814, 0.039568];
    bias_6 : ARRAY[0..21] OF REAL := [-0.038554, -0.069090, -0.070693, -0.115084, -0.097080, -0.129611, -0.166989, -0.007479, -0.116594, -0.036034, -0.019034, -0.083656, -0.060446, -0.028157, -0.117170, -0.144152, -0.075183, -0.087516, -0.057288, 0.007025, -0.044599, -0.069669];

    weights_7 : ARRAY[0..483] OF REAL := [-0.364807, -0.237205, 0.003107, -0.277985, -0.266964, 0.229299, 0.226449, -0.115922, 0.346281, -0.122565, -0.071139, 0.316857, -0.253779, 0.083801, -0.321255, 0.213799, 0.367622, 0.011978, -0.192643, -0.374560, 0.056494, 0.148061, 0.035985, -0.165501, -0.210764, 0.217239, -0.027652, 0.241365, -0.133801, -0.107932, -0.177462, 0.233720, 0.209747, -0.214530, 0.217923, -0.349102, 0.359582, 0.204399, 0.304146, 0.248734, 0.067950, -0.219972, -0.099247, 0.283676, -0.233460, 0.309059, 0.182080, 0.321843, -0.042071, 0.197389, 0.140214, 0.241827, 0.085037, 0.109508, -0.220502, -0.220265, -0.087820, -0.119139, 0.323995, -0.122659, -0.214543, -0.031225, -0.220536, -0.084045, 0.342094, -0.304938, -0.166558, -0.331302, -0.034692, -0.070936, 0.374081, -0.000861, -0.055461, 0.245237, -0.093936, 0.094637, -0.252934, -0.270222, 0.239100, -0.094572, 0.085492, 0.152916, 0.147673, 0.339831, -0.148906, 0.272575, 0.226315, 0.178353, -0.004990, -0.017697, 0.269839, 0.076927, -0.062259, 0.329724, 0.162755, -0.175503, 0.174239, -0.355379, -0.200217, 0.321982, 0.312672, -0.100468, -0.239923, -0.306172, 0.311937, -0.041929, 0.068473, -0.002791, 0.310846, -0.262511, 0.000795, 0.076557, -0.296009, 0.360625, -0.096104, -0.048972, 0.035857, -0.129680, 0.285704, -0.065346, -0.193558, -0.020755, 0.243402, 0.406058, -0.293829, -0.074964, -0.145684, 0.211279, 0.349128, -0.247246, 0.245466, -0.187025, 0.132599, -0.021370, 0.238913, 0.070160, 0.026178, 0.289003, 0.128294, 0.286053, 0.048953, 0.144959, -0.165488, 0.129873, 0.237547, -0.123310, -0.018060, -0.023911, -0.181706, 0.232393, 0.004010, -0.235293, -0.358987, -0.267835, -0.087012, -0.038157, 0.386318, 0.282579, -0.269643, -0.204573, -0.118866, -0.103115, -0.159380, 0.412627, 0.039357, 0.409754, 0.367476, 0.199884, -0.033722, -0.072961, 0.156928, -0.157388, 0.090366, 0.247479, 0.245104, 0.027052, 0.225238, 0.052037, 0.371539, 0.091238, 0.052721, 0.379377, -0.108780, 0.078507, -0.183822, 0.217486, 0.126594, -0.213494, -0.061266, 0.066101, 0.315268, -0.155193, -0.029315, -0.034761, 0.157296, -0.104517, -0.100141, -0.294797, 0.288260, -0.169811, -0.303266, -0.082669, 0.148466, 0.081710, 0.316547, -0.152269, 0.184802, 0.146022, 0.096096, 0.002435, -0.295222, -0.269055, -0.195022, 0.277882, 0.026990, -0.076466, -0.210177, 0.147231, -0.333660, 0.020189, 0.183079, -0.016232, -0.067070, -0.252107, 0.327201, -0.205255, -0.043016, -0.201926, -0.208554, -0.013192, 0.253420, -0.007254, -0.279261, -0.131021, 0.371989, 0.144509, 0.300232, -0.036232, -0.049781, -0.044779, 0.188152, -0.103627, -0.272634, -0.126766, 0.228000, -0.218025, -0.275888, 0.229057, 0.296634, -0.299150, -0.025997, -0.153610, 0.077227, 0.144796, -0.135159, -0.171910, 0.348851, 0.323723, 0.059755, -0.320430, -0.299073, -0.186415, 0.200756, 0.371905, 0.045845, -0.059686, -0.075543, 0.175812, 0.069348, 0.044875, 0.008746, -0.336807, 0.284989, 0.011657, -0.156655, -0.117098, -0.334991, 0.178509, 0.233031, -0.346055, -0.020197, -0.338296, -0.121066, -0.009821, 0.090784, 0.233949, -0.055547, -0.321706, -0.187452, -0.105880, 0.146602, 0.072494, 0.267509, -0.049071, -0.193850, 0.284649, -0.285856, -0.147783, -0.278323, 0.155102, 0.382837, 0.088352, 0.300924, 0.265163, 0.059495, -0.000278, -0.258798, -0.352332, -0.064502, 0.272706, -0.101842, 0.116434, 0.393129, -0.195981, 0.171106, -0.163257, 0.312684, 0.257203, 0.038465, 0.251090, -0.317675, -0.009819, 0.100809, 0.015764, -0.217878, 0.276626, 0.273479, -0.068491, -0.177248, -0.200985, 0.021487, 0.310245, 0.140616, -0.186077, 0.237085, 0.272650, -0.238218, -0.193871, 0.030906, 0.172769, 0.206835, -0.367597, 0.111000, -0.114181, 0.014274, 0.157484, 0.182549, -0.212528, -0.159400, 0.068230, 0.105951, 0.122735, 0.077816, -0.205018, -0.103166, -0.298082, 0.087485, 0.035753, 0.328822, 0.314977, -0.264400, -0.011742, 0.145015, -0.228218, 0.100806, -0.070884, -0.160237, 0.288215, -0.121132, 0.235051, -0.182789, -0.048591, -0.364731, 0.292513, -0.099273, -0.349288, 0.162773, 0.178850, 0.019613, 0.052627, 0.365623, -0.144881, -0.351180, -0.337891, -0.212585, 0.112071, -0.346731, -0.249420, 0.296264, 0.201225, -0.095385, -0.098909, 0.261799, 0.307101, 0.273750, 0.108290, -0.083510, 0.295069, -0.112469, -0.209436, 0.220792, 0.109743, -0.065429, 0.034753, 0.248463, -0.172492, 0.070443, -0.002859, 0.241954, -0.081209, 0.089796, 0.067934, 0.123482, -0.059438, -0.160759, -0.000107, 0.033234, 0.372172, -0.278811, 0.260340, -0.015133, 0.271877, -0.132613, -0.210920, 0.153416, -0.117573, -0.109628, -0.034458, -0.318392, -0.299637, 0.161219, 0.144702, -0.228644, -0.083063, -0.274778, -0.157896, -0.175295, 0.201361, -0.162565, -0.086850, 0.280234, 0.239699, -0.205100, -0.007323, -0.263147, -0.160285, 0.036830, 0.188243, -0.025224, -0.047957, 0.135811, -0.284034, 0.208566, 0.196352, 0.121749, 0.217313, 0.250076, 0.153696, -0.269822, 0.033041, -0.321990, -0.200328, 0.383204, 0.298319, 0.356129, 0.164212, 0.354779, 0.122489, -0.277260, 0.306636, 0.110841, -0.194020, -0.232883, -0.243732, 0.065778, -0.187497, -0.057630, 0.271607, 0.160529, -0.381793, 0.077020, 0.313479, 0.164137, 0.229028];
    bias_7 : ARRAY[0..21] OF REAL := [0.004210, -0.065403, -0.038060, -0.009318, 0.002655, -0.043196, -0.088895, -0.065542, -0.058176, -0.060855, -0.012981, -0.104761, -0.045089, -0.031662, -0.070532, -0.028477, -0.031021, -0.067918, -0.042964, -0.073024, -0.086002, -0.020363];

    weights_8 : ARRAY[0..483] OF REAL := [-0.304101, 0.100405, 0.002995, 0.057810, -0.242602, -0.273599, -0.121230, -0.334182, 0.093236, 0.325720, -0.074310, -0.055977, -0.036704, 0.217162, 0.217684, -0.148756, -0.161542, -0.331079, 0.336452, 0.002076, 0.064254, -0.285264, 0.004341, -0.190827, 0.115994, 0.179272, -0.221798, 0.154819, -0.051903, 0.007554, -0.126661, -0.308765, 0.084443, -0.156972, -0.024309, 0.035879, 0.270818, -0.016274, 0.251293, -0.028767, 0.315917, -0.001414, 0.316582, -0.119401, -0.190033, -0.275479, -0.013381, -0.370872, -0.206311, -0.281223, -0.293913, 0.075550, -0.150843, -0.217919, -0.030059, 0.312021, 0.186389, 0.125019, -0.025959, -0.025464, -0.294949, 0.332481, 0.131844, 0.101673, -0.013060, 0.207647, -0.256493, -0.212812, -0.376007, 0.201892, 0.112231, -0.286955, 0.104312, 0.190116, 0.052606, -0.267054, 0.291532, -0.089247, -0.136573, -0.206726, -0.024356, -0.189374, -0.001127, -0.313542, 0.274362, -0.203525, 0.323169, -0.100039, 0.132450, -0.151800, -0.220307, 0.112444, -0.049819, 0.122316, 0.000369, 0.111705, 0.088284, 0.049253, 0.242499, -0.286597, -0.361232, -0.163359, -0.320030, -0.020116, -0.326576, -0.118994, -0.120750, -0.151636, 0.312837, 0.280238, 0.124667, -0.112507, 0.222865, -0.073986, 0.244271, 0.034561, 0.024196, 0.103750, -0.260433, 0.325997, -0.030559, -0.029249, -0.171641, -0.253439, -0.227437, -0.336349, 0.107598, -0.117105, -0.148553, -0.238698, 0.109604, 0.365084, -0.114405, 0.101671, 0.038573, -0.067465, -0.255861, -0.306121, 0.339633, -0.049495, 0.217593, -0.050345, 0.325784, -0.006173, -0.162129, 0.343760, -0.037653, -0.060563, 0.154156, -0.244862, 0.027071, 0.312544, -0.133437, 0.234843, 0.197283, 0.018649, 0.037359, 0.188100, -0.286412, 0.060599, 0.339736, 0.361118, -0.008767, -0.031222, -0.222021, 0.272277, -0.146847, -0.066719, 0.010102, -0.303984, 0.265519, -0.180363, 0.210170, -0.235923, 0.137099, 0.067770, -0.084659, 0.048161, -0.193153, 0.194766, 0.174274, 0.189377, -0.374807, -0.097780, 0.090249, 0.339279, 0.113975, -0.174171, -0.379416, -0.053263, 0.215209, -0.060534, -0.063412, -0.178798, -0.163625, -0.110166, 0.353055, 0.032388, 0.021996, -0.067057, 0.322100, 0.097297, 0.279732, -0.095723, -0.256106, -0.218846, 0.079269, -0.201426, -0.109792, 0.058115, 0.100504, 0.128473, 0.055302, -0.251147, -0.349522, 0.326949, -0.150755, -0.258978, 0.350044, 0.368011, 0.102035, -0.075404, -0.153538, 0.039335, -0.199097, -0.066225, -0.273895, -0.299174, 0.150867, 0.326326, 0.093391, -0.369773, 0.025218, 0.116055, 0.298750, -0.107689, -0.021658, -0.182893, -0.164422, -0.375683, 0.238609, -0.014968, -0.059321, 0.271235, 0.295513, 0.243225, -0.355273, -0.184175, 0.126072, -0.020273, -0.368423, -0.292870, -0.119282, 0.214852, -0.308788, -0.156068, 0.005302, -0.048743, 0.118361, 0.362293, -0.206345, 0.392740, -0.077161, -0.049853, -0.080545, -0.399856, 0.320488, -0.127193, 0.338027, -0.346031, -0.079254, 0.043530, -0.068631, 0.015204, 0.002581, -0.226777, -0.416716, 0.302243, 0.050058, 0.251215, -0.150563, -0.007115, -0.096752, -0.318998, 0.119210, -0.128624, 0.418948, 0.281796, -0.290408, -0.310466, -0.176446, -0.225991, -0.244705, 0.184350, 0.154406, 0.172996, 0.221570, 0.353859, -0.245753, -0.052207, 0.345642, -0.117925, 0.110679, 0.237876, -0.302092, 0.128750, 0.179905, -0.118239, 0.192334, 0.062414, -0.277213, 0.269299, -0.107412, -0.044930, 0.101491, 0.142444, -0.075570, -0.068008, 0.288095, 0.290121, -0.358004, 0.150708, -0.352893, -0.162085, -0.257908, 0.116579, 0.317240, -0.181375, -0.121135, -0.294720, -0.336578, 0.258292, -0.017588, 0.272614, -0.145503, -0.363242, 0.117636, -0.330467, -0.088475, -0.272619, 0.012840, 0.335567, 0.197085, -0.264906, -0.117633, -0.165108, 0.167619, 0.088469, -0.228842, -0.215362, 0.341731, 0.236351, 0.139205, 0.034800, 0.061918, -0.209297, 0.041870, 0.233346, -0.031528, 0.329038, 0.127629, 0.095076, 0.125804, 0.253046, -0.348896, 0.326187, 0.109988, 0.140123, -0.023594, 0.150104, 0.264505, 0.294146, 0.075023, 0.258969, -0.306224, -0.174115, -0.123953, -0.201984, -0.323234, -0.263548, -0.091933, 0.164536, 0.235985, -0.114475, 0.006051, -0.321960, -0.238489, -0.338807, 0.273570, 0.034605, 0.048560, 0.257436, 0.237913, 0.100005, -0.193065, 0.135461, -0.225799, -0.240579, -0.321482, -0.191338, 0.235546, -0.052109, -0.310213, 0.023116, -0.330784, 0.002633, 0.029876, 0.086963, -0.225957, -0.105181, 0.186328, 0.108465, 0.102253, 0.071713, 0.104452, -0.022872, -0.093682, 0.348286, 0.122766, -0.291970, -0.077946, -0.026091, 0.049628, 0.275843, 0.304503, -0.064878, -0.101381, 0.141398, 0.312967, -0.061732, -0.168198, -0.087561, 0.019208, -0.216387, -0.245466, 0.335886, -0.209319, -0.211301, 0.254174, -0.108969, 0.107924, 0.125145, -0.005004, 0.151247, -0.220327, -0.263631, -0.125216, -0.065397, 0.089067, 0.038949, 0.288617, -0.074407, -0.146795, 0.365915, 0.129221, 0.033395, 0.015230, 0.183953, 0.074455, -0.043828, -0.045802, -0.269612, -0.100710, -0.366374, -0.204745, -0.338251, 0.248442, -0.335265, 0.036204, -0.352897, -0.125164, -0.006339, 0.148360, -0.353406, 0.126088, 0.160982, -0.174683, 0.004713, 0.076501, 0.053836, 0.010805, 0.149345, 0.241343, -0.017611];
    bias_8 : ARRAY[0..21] OF REAL := [-0.053942, -0.039806, -0.114276, -0.077186, -0.108063, 0.138418, -0.045914, -0.113785, -0.090467, 0.002213, -0.001533, -0.066077, -0.034647, -0.006248, -0.109403, -0.049483, -0.029343, -0.048922, -0.009135, 0.062359, -0.002033, -0.010056];

    weights_9 : ARRAY[0..483] OF REAL := [0.291405, 0.141374, 0.282357, -0.077351, -0.041122, 0.044482, -0.177353, 0.033180, 0.117982, 0.244526, 0.322031, -0.044921, -0.053637, 0.280691, 0.239119, 0.191502, 0.111717, 0.032084, -0.361666, 0.155028, 0.170054, 0.167260, 0.188853, -0.252937, -0.295169, 0.195733, 0.165755, 0.190833, 0.197284, -0.137282, -0.021825, -0.080116, 0.312367, -0.096758, 0.293003, 0.054252, -0.019322, -0.187552, 0.155657, 0.015608, 0.167133, 0.025319, -0.081355, 0.260660, 0.291596, 0.317451, 0.064761, -0.079913, 0.078364, 0.101550, 0.291632, 0.039102, 0.308560, -0.348539, 0.197361, 0.028542, -0.055312, -0.121961, 0.157019, -0.389426, 0.083265, 0.268963, -0.268128, -0.040137, -0.362593, -0.303184, 0.258013, 0.216494, 0.330328, 0.309907, 0.311888, 0.180359, -0.266960, -0.068229, -0.309373, 0.238089, 0.209288, -0.123857, -0.125822, -0.355802, 0.052387, 0.186312, 0.351722, 0.330626, -0.116407, -0.214591, -0.096964, 0.103042, -0.139619, 0.137578, 0.238847, 0.196291, -0.203072, -0.022230, 0.043055, -0.310298, -0.148519, 0.149099, 0.192962, 0.265896, 0.247786, 0.070531, -0.277392, 0.080622, 0.069952, 0.301300, -0.283804, -0.025043, 0.023874, 0.207036, 0.278743, -0.138272, 0.072829, 0.133706, -0.168225, 0.236182, 0.186555, 0.259680, 0.056683, -0.355899, -0.062051, 0.031430, 0.398269, 0.370913, 0.306754, 0.241362, 0.092240, -0.333993, 0.232807, -0.035876, 0.018400, 0.068558, 0.144214, 0.006177, 0.316347, 0.154232, -0.262014, -0.324933, -0.184725, 0.217085, 0.333744, 0.106959, -0.188327, 0.115254, 0.007724, 0.226681, -0.309198, -0.137253, -0.126305, -0.194801, 0.065863, -0.149419, -0.264038, -0.158259, 0.100875, -0.195858, -0.028089, 0.023821, 0.065104, 0.013864, 0.056584, -0.348344, -0.102075, 0.271184, -0.337538, -0.122690, 0.260882, 0.228452, 0.322926, -0.087738, -0.067590, 0.187356, 0.052459, 0.364149, -0.127055, -0.316370, 0.281382, 0.063545, 0.327750, 0.230121, 0.240535, 0.105809, 0.049031, -0.208946, -0.102982, -0.217016, 0.052294, -0.111517, 0.102462, -0.035382, -0.126871, 0.003332, 0.302876, -0.187831, 0.162267, 0.206348, 0.123683, 0.178614, -0.195703, -0.138148, 0.136203, -0.141306, -0.242701, 0.118960, 0.248093, 0.085925, -0.043043, -0.096688, 0.320477, 0.256843, -0.281589, -0.289960, 0.106101, -0.033407, 0.149314, 0.184856, -0.065799, 0.230886, -0.108866, 0.250446, -0.156062, -0.131783, 0.190123, 0.010329, 0.042087, 0.075380, -0.380883, 0.256218, 0.285787, -0.000133, 0.273594, 0.295604, -0.059781, -0.342750, -0.055721, -0.247609, -0.336659, 0.147422, 0.131190, 0.010688, -0.105754, -0.391031, -0.287063, -0.021181, -0.318998, 0.107840, -0.149239, 0.262757, -0.214663, -0.129526, -0.164720, 0.307621, -0.341077, -0.165969, -0.323687, 0.371293, 0.332246, -0.336607, -0.085555, 0.379451, -0.254800, -0.031013, 0.093902, 0.211159, 0.101238, -0.353260, -0.301462, -0.200904, 0.154387, -0.104396, -0.193023, -0.007422, -0.145247, -0.203819, 0.242737, 0.108415, -0.006407, -0.098772, 0.013168, -0.351755, -0.012058, -0.109795, -0.269478, 0.116324, 0.065023, -0.249584, 0.254341, -0.321049, -0.241100, -0.253269, -0.223128, 0.327500, 0.195053, 0.105591, 0.152155, -0.070858, 0.103443, 0.121845, -0.231868, -0.239906, 0.345326, -0.139534, 0.320864, 0.152868, 0.040831, 0.307245, 0.147165, 0.211801, 0.212192, -0.142130, 0.290436, 0.287465, 0.021244, 0.301013, 0.243155, 0.189223, 0.267868, -0.000688, -0.356680, -0.143016, -0.303536, 0.121200, 0.251932, -0.130832, 0.054976, -0.276335, 0.025617, -0.085358, -0.045851, -0.248477, 0.255845, 0.366110, -0.148382, 0.249056, 0.031657, -0.139340, -0.127775, 0.369570, -0.078088, 0.136977, -0.243397, -0.169195, -0.249370, 0.276968, -0.247236, 0.233353, 0.302598, -0.107487, -0.053783, 0.322470, 0.328018, -0.136053, 0.179077, 0.189144, 0.115060, 0.292244, -0.094431, 0.025864, 0.145910, 0.272067, 0.139002, 0.188885, -0.299509, 0.197325, 0.036821, 0.134966, 0.141116, 0.273156, -0.073848, -0.310700, 0.241425, -0.073763, -0.156702, 0.300883, -0.084753, -0.172269, 0.213301, 0.200072, 0.386469, 0.268827, -0.048445, -0.252957, -0.099254, 0.177895, -0.080412, -0.057002, -0.246679, -0.164205, 0.223254, 0.108977, 0.159682, 0.226258, 0.179821, -0.051758, -0.089191, -0.246040, 0.319253, 0.174879, -0.184168, -0.239251, 0.135208, 0.107313, 0.147043, 0.064580, 0.344720, 0.267251, 0.154827, 0.332723, 0.264895, -0.036242, -0.203609, -0.345307, 0.201927, -0.195573, 0.323279, 0.218110, -0.333786, 0.108415, -0.036261, 0.246995, 0.121394, 0.058787, 0.400554, -0.196602, 0.299842, -0.175333, 0.342154, -0.184092, 0.006567, -0.227063, 0.280483, 0.348923, -0.211455, -0.347464, 0.173309, 0.232733, -0.168795, 0.244171, -0.050568, 0.275496, 0.053077, 0.126551, -0.226761, -0.002516, -0.088065, 0.017988, -0.459883, 0.017205, -0.006719, -0.192900, -0.403844, 0.197305, -0.273246, 0.181749, -0.389882, -0.034637, 0.264911, 0.178060, -0.337430, 0.275195, -0.285267, 0.114618, 0.210708, 0.345090, 0.115794, -0.116793, 0.240980, -0.329921, 0.023980, -0.314724, 0.292355, 0.129115, -0.134935, 0.272835, -0.020539, -0.232311, -0.122839, 0.099400, -0.280323, -0.107125, -0.237164, 0.097858, -0.242950, 0.001372];
    bias_9 : ARRAY[0..21] OF REAL := [-0.042123, 0.000777, -0.111340, -0.027852, -0.033235, -0.019487, 0.334357, -0.034739, -0.027430, 0.022708, -0.013594, 0.010036, 0.288000, 0.195808, -0.040669, -0.117542, -0.117658, -0.052323, 0.313272, -0.018863, -0.050297, -0.029875];

    weights_10 : ARRAY[0..483] OF REAL := [-0.349085, -0.255252, -0.405605, -0.254197, -0.085029, 0.154930, -0.181518, -0.167803, -0.132807, -0.248886, 0.010728, 0.052639, -0.426656, 0.040061, -0.143751, 0.272906, 0.251352, -0.262541, -0.360687, -0.093133, -0.028936, 0.127721, -0.332217, 0.175673, 0.193391, -0.399545, -0.166332, -0.146595, -0.311122, -0.376500, 0.038709, -0.072278, -0.285064, -0.165089, 0.151159, -0.066235, 0.044413, 0.170296, -0.207504, 0.431780, -0.472849, 0.114538, 0.112523, -0.372727, 0.017929, 0.283571, -0.441509, 0.000893, 0.142533, -0.148300, 0.234689, -0.153648, -0.262494, -0.015331, 0.319015, -0.194357, 0.098355, 0.302037, 0.269415, -0.109922, 0.129879, -0.165909, -0.490637, 0.242059, 0.240485, 0.240986, 0.214114, 0.169973, -0.487652, 0.246876, -0.092630, 0.218701, 0.172268, -0.184838, 0.210873, -0.221048, 0.052754, 0.276413, 0.039480, 0.245392, 0.220094, 0.235335, -0.320727, -0.137810, 0.268048, 0.144431, -0.017521, -0.185173, -0.060579, 0.028087, -0.257993, 0.064159, -0.371356, 0.135866, 0.030787, 0.147261, -0.365286, 0.200039, -0.069716, -0.107996, -0.276796, 0.138753, 0.368345, 0.332594, 0.022675, -0.077018, -0.407025, -0.375562, 0.174454, 0.184695, -0.069322, -0.114921, -0.071543, -0.268611, -0.043742, 0.112823, 0.325665, -0.189783, 0.292052, 0.006862, 0.234574, 0.108378, -0.115613, 0.369941, -0.071301, 0.307281, -0.072362, 0.093566, 0.039918, 0.129114, 0.298354, -0.190702, 0.120265, 0.305333, 0.183508, -0.331026, -0.099257, 0.049817, -0.275575, -0.026829, -0.345661, -0.377555, 0.141504, -0.001494, 0.345864, -0.069530, 0.159165, 0.245421, -0.284704, 0.222901, 0.192191, -0.169666, 0.078370, 0.311888, -0.138020, -0.265656, -0.474406, 0.341808, 0.031872, -0.201934, -0.152700, -0.138257, -0.356230, 0.007561, 0.120031, -0.354471, -0.355637, -0.089398, 0.274328, 0.082394, 0.123461, -0.140907, -0.241772, 0.225848, 0.165791, 0.253905, 0.198775, -0.039124, 0.156383, 0.215096, 0.209061, -0.338914, -0.213092, -0.157497, -0.038457, -0.324363, -0.284082, -0.345515, -0.431152, 0.338202, 0.021150, 0.164488, 0.219146, -0.070000, -0.480418, 0.114832, 0.066806, -0.050485, 0.112560, -0.372389, -0.556418, -0.219756, -0.155614, 0.215980, -0.157124, -0.091571, -0.037490, 0.207084, 0.177779, 0.099052, -0.063657, 0.029919, 0.364368, 0.427587, 0.114253, 0.241202, -0.244599, 0.156045, -0.070967, -0.089008, -0.261334, 0.006399, -0.026032, -0.420007, -0.272231, 0.090441, -0.227075, -0.166100, 0.304352, 0.252615, -0.060726, -0.084069, 0.135438, 0.198651, -0.154068, 0.134615, 0.347210, 0.277948, -0.467889, -0.298930, 0.038240, -0.219938, -0.281739, 0.215830, -0.381041, -0.030534, -0.286199, -0.432523, -0.214966, 0.134648, -0.115906, -0.339068, -0.407640, -0.116214, -0.571897, 0.150820, -0.011836, 0.319152, 0.058787, -0.051251, -0.008618, -0.239970, -0.156657, -0.326832, 0.195360, 0.303078, 0.139692, -0.151020, 0.292342, -0.292876, 0.117475, -0.038759, -0.298126, 0.183821, 0.128326, 0.126459, 0.308505, 0.232574, -0.245094, -0.272323, 0.059468, -0.093050, 0.396356, 0.244080, -0.113235, -0.014609, 0.282617, 0.099241, 0.485838, 0.324977, -0.041194, -0.223290, 0.347672, -0.080127, 0.162102, -0.034238, 0.243998, 0.094273, 0.320944, 0.291878, 0.037718, 0.355247, -0.212855, -0.325569, 0.053696, -0.124852, 0.289413, 0.277775, 0.102272, -0.014392, -0.299137, 0.184444, 0.227217, 0.094097, 0.235190, -0.179700, 0.055732, -0.257083, -0.218430, 0.213285, 0.155567, -0.157689, 0.031142, 0.192005, 0.161268, -0.005469, 0.228666, 0.119225, 0.304275, -0.289531, -0.073998, 0.203284, 0.081919, -0.090304, 0.060548, 0.275761, 0.358002, 0.267586, 0.068037, 0.209190, 0.128446, 0.257392, 0.175913, -0.293333, 0.167319, -0.279665, 0.119015, -0.132297, -0.281729, -0.123650, 0.152962, 0.052877, -0.126414, -0.055418, -0.392282, -0.283558, -0.155702, -0.113843, 0.295736, 0.030909, -0.004687, -0.025172, -0.283908, -0.090191, 0.171230, -0.192925, -0.189608, -0.128366, 0.425038, 0.122842, -0.243712, -0.323571, 0.086517, 0.187092, -0.337402, -0.325973, -0.492802, -0.002252, -0.195425, 0.031600, 0.240169, -0.425103, 0.009069, -0.184859, -0.322816, -0.184279, 0.174795, 0.191188, 0.285365, 0.243636, 0.305782, -0.264094, -0.076863, -0.275164, 0.091100, 0.041269, 0.061536, -0.055633, 0.243271, -0.233997, -0.010786, -0.031630, 0.168606, 0.260526, -0.356548, 0.013765, -0.150032, -0.354842, 0.160712, -0.219600, 0.052887, -0.021269, 0.342403, -0.259443, 0.416458, -0.274569, -0.005679, 0.296961, -0.033346, -0.132873, -0.504612, -0.019323, 0.079945, -0.162185, 0.057476, -0.306967, -0.414108, 0.124638, -0.004922, -0.072289, -0.170029, 0.184850, 0.083754, 0.100674, -0.356607, 0.460382, -0.714262, -0.363000, 0.363790, -0.245974, -0.144517, 0.133035, 0.291362, -0.375774, -0.004475, 0.129743, 0.309834, -0.131199, 0.126412, -0.105008, -0.073435, -0.210801, 0.186747, 0.001864, -0.324538, 0.123541, 0.076056, 0.247461, 0.099651, 0.338382, 0.283419, -0.184649, -0.169476, -0.325189, -0.430024, 0.313859, -0.202028, 0.165602, -0.052410, 0.175244, -0.101641, 0.031976, -0.101026, 0.255282, -0.338211, 0.076702, -0.026419, 0.015351, 0.095367, -0.103350, -0.290732, -0.386126, 0.105620, 0.110101];
    bias_10 : ARRAY[0..21] OF REAL := [-0.244935, 0.078022, 0.535524, 0.222739, 0.112724, -0.118234, -0.143530, -0.140477, -0.097571, -0.135936, 0.237141, -0.079870, 0.299600, -0.080816, -0.102707, -0.093236, -0.128525, 0.059616, 0.479920, -0.000087, -0.093376, 0.247937];

    weights_11 : ARRAY[0..65] OF REAL := [-0.262914, 0.217390, -0.032490, -0.038667, -0.222139, -0.108030, 0.840270, -0.271333, -0.403203, -0.110824, 0.032260, -0.143203, -0.026281, -0.396157, -0.159642, -0.234800, 0.281971, -0.403431, -0.163432, -0.353595, 0.180655, -0.077111, 0.287310, -0.368344, 0.330888, 0.425896, -0.329624, 0.084356, -0.002153, -0.359770, 0.430353, -0.256014, 0.082786, -0.385118, 0.056951, -0.184230, 0.461194, -0.169245, -0.020006, -0.178489, 0.157042, 0.348702, -0.411279, -0.166043, 0.275035, -0.305084, 0.266472, 0.362730, -0.269294, -0.255215, 0.116720, -0.243887, 0.300924, 0.466904, 0.589079, -0.570996, -0.484486, -0.316679, 0.096183, -0.264100, -0.248617, 0.069060, 0.434102, 0.093867, -0.397841, -0.443745];
    bias_11 : ARRAY[0..2] OF REAL := [0.207550, 0.163853, -0.315461];

END_VAR

VAR
    (* Buffer allocation variables *)
    buffer_0 : ARRAY[0..21] OF REAL;
    buffer_1 : ARRAY[0..21] OF REAL;

    (* Temporary computation variables *)
    i : DINT;
    j : DINT;
    sum : REAL;
    max_val : REAL;
    exp_sum : REAL;

END_VAR

(* Layer 0: Fused Linear + RELU *)
FOR j := 0 TO 21 DO
    sum := 0.0;
    FOR i := 0 TO 4 DO
        sum := sum + input_data[i] * weights_0[i * 22 + j];
    END_FOR;
    buffer_1[j] := MAX(sum + bias_0[j], 0.0);
END_FOR;

(* Layer 1: Fused Linear + RELU *)
FOR j := 0 TO 21 DO
    sum := 0.0;
    FOR i := 0 TO 21 DO
        sum := sum + buffer_1[i] * weights_1[i * 22 + j];
    END_FOR;
    buffer_0[j] := MAX(sum + bias_1[j], 0.0);
END_FOR;

(* Layer 2: Fused Linear + RELU *)
FOR j := 0 TO 21 DO
    sum := 0.0;
    FOR i := 0 TO 21 DO
        sum := sum + buffer_0[i] * weights_2[i * 22 + j];
    END_FOR;
    buffer_1[j] := MAX(sum + bias_2[j], 0.0);
END_FOR;

(* Layer 3: Fused Linear + RELU *)
FOR j := 0 TO 21 DO
    sum := 0.0;
    FOR i := 0 TO 21 DO
        sum := sum + buffer_1[i] * weights_3[i * 22 + j];
    END_FOR;
    buffer_0[j] := MAX(sum + bias_3[j], 0.0);
END_FOR;

(* Layer 4: Fused Linear + RELU *)
FOR j := 0 TO 21 DO
    sum := 0.0;
    FOR i := 0 TO 21 DO
        sum := sum + buffer_0[i] * weights_4[i * 22 + j];
    END_FOR;
    buffer_1[j] := MAX(sum + bias_4[j], 0.0);
END_FOR;

(* Layer 5: Fused Linear + RELU *)
FOR j := 0 TO 21 DO
    sum := 0.0;
    FOR i := 0 TO 21 DO
        sum := sum + buffer_1[i] * weights_5[i * 22 + j];
    END_FOR;
    buffer_0[j] := MAX(sum + bias_5[j], 0.0);
END_FOR;

(* Layer 6: Fused Linear + RELU *)
FOR j := 0 TO 21 DO
    sum := 0.0;
    FOR i := 0 TO 21 DO
        sum := sum + buffer_0[i] * weights_6[i * 22 + j];
    END_FOR;
    buffer_1[j] := MAX(sum + bias_6[j], 0.0);
END_FOR;

(* Layer 7: Fused Linear + RELU *)
FOR j := 0 TO 21 DO
    sum := 0.0;
    FOR i := 0 TO 21 DO
        sum := sum + buffer_1[i] * weights_7[i * 22 + j];
    END_FOR;
    buffer_0[j] := MAX(sum + bias_7[j], 0.0);
END_FOR;

(* Layer 8: Fused Linear + RELU *)
FOR j := 0 TO 21 DO
    sum := 0.0;
    FOR i := 0 TO 21 DO
        sum := sum + buffer_0[i] * weights_8[i * 22 + j];
    END_FOR;
    buffer_1[j] := MAX(sum + bias_8[j], 0.0);
END_FOR;

(* Layer 9: Fused Linear + RELU *)
FOR j := 0 TO 21 DO
    sum := 0.0;
    FOR i := 0 TO 21 DO
        sum := sum + buffer_1[i] * weights_9[i * 22 + j];
    END_FOR;
    buffer_0[j] := MAX(sum + bias_9[j], 0.0);
END_FOR;

(* Layer 10: Fused Linear + RELU *)
FOR j := 0 TO 21 DO
    sum := 0.0;
    FOR i := 0 TO 21 DO
        sum := sum + buffer_0[i] * weights_10[i * 22 + j];
    END_FOR;
    buffer_1[j] := MAX(sum + bias_10[j], 0.0);
END_FOR;

(* Layer 11: Fused Linear + SOFTMAX *)
FOR j := 0 TO 2 DO
    sum := 0.0;
    FOR i := 0 TO 21 DO
        sum := sum + buffer_1[i] * weights_11[i * 3 + j];
    END_FOR;
    output_data[j] := sum + bias_11[j];
END_FOR;

max_val := output_data[0];
FOR i := 1 TO 2 DO
    IF output_data[i] > max_val THEN
        max_val := output_data[i];
    END_IF;
END_FOR;

exp_sum := 0.0;
FOR i := 0 TO 2 DO
    output_data[i] := EXP(output_data[i] - max_val);
    exp_sum := exp_sum + output_data[i];
END_FOR;

FOR i := 0 TO 2 DO
    output_data[i] := output_data[i] / exp_sum;
END_FOR;

END_FUNCTION_BLOCK
